{attribute 'qualified_only' := ''}
{attribute 'strict' := ''}
TYPE eFirmerVendorEvent3 :
(
	eNoInfo := 0,
	eFanFault := 1,
	eStatisticsMemoryFault := 2,
	eRTCClockNotSet := 3,
	eRTCLowBatteryFault := 5,
	eRTCQuartzFault := 6
);
END_TYPE

(* stored: Version 1.1.0.1, ProductVersion 3.1.4024.11
   DUT eFirmerVendorEvent3: Id {102bce57-bb61-4765-9dee-df1847233910} *)
